Fanuc KAREL source: CA0109.KL

-- PROVISIONAL review KL for V1013-1; original PC SHA256 76fd3dc815e8e102fc7612b9a437d29ec366bbab3dc83c6857e579deb10c6ad6
-- Incomplete behavior may be omitted. Consult companion uncertainty JSON. Do not deploy.
PROGRAM CA0109
%NOLOCKGROUP
BEGIN
  -- UNRESOLVED_PC offsets 0-1; opcodes 7B
  -- UNRESOLVED_PC offsets 6-18; opcodes 2D,9D,52,7F
  -- UNRESOLVED_PC offsets 23-27; opcodes 7F
  -- UNRESOLVED_PC offsets 32-39; opcodes 9C,23
  -- UNRESOLVED_PC offsets 44-51; opcodes 9D,23
  -- UNRESOLVED_PC offsets 56-67; opcodes 2E,23
  -- UNRESOLVED_PC offsets 72-79; opcodes 9D,23
  -- UNRESOLVED_PC offsets 84-93; opcodes 3F,75
  -- UNRESOLVED_PC offsets 98-112; opcodes 2E,22,9D,33,35
  -- UNRESOLVED_PC offsets 117-131; opcodes 2E,22,9D,33,35
  -- UNRESOLVED_PC offsets 136-151; opcodes 2E,22,32,35
  -- UNRESOLVED_PC offsets 156-171; opcodes 2E,22,32,35
  -- UNRESOLVED_PC offsets 176-198; opcodes 27,22,AA,2E,52,23
  -- UNRESOLVED_PC offsets 203-207; opcodes 7F
END CA0109
